# EPICS substitutions: Module_7_EPICS_databases/FirstAirCondSys/FirstACApp/Db/ACSys.substitutions
# Air Conditioning System substitutions file

file "db/dbAirCondSys.db" {
    { user = "codac-dev", InsulCoeff = 0.02, HighTmp = 30, LowTmp = 25, PreSetTmp = 22, DeadBand = 0.2, Power = 0.4 }
}
